FUNCTION_BLOCK FB_LowerFeedInConveyor EXTENDS FB_ActionBasic
VAR_INPUT
    xExecute    : BOOL;
    xAbort      : BOOL;
	xReset		: BOOL;
    Cylinder 	: REFERENCE TO UNI_CylinderList;
    TimeOut  	: LREAL := 30; // Unit : s
	Input		: ST_InputTable;
	OutPut		: ST_OutputTable;
	Motor		: REFERENCE TO UNI_MotorList;
END_VAR	
VAR_OUTPUT
    xAborted : BOOL;
    iErrorID : INT;
    ErrorMsg : T_MaxString;
END_VAR
VAR
    StateBehaviour   : CBML.ETrigATo;
    CurrentPosition : ST_PositionTable;
	uiCyclicStep    : UINT := 0;
	Reset_Rtrig 	:R_TRIG;
	
	TON_SensorDelay :TON;
	TON_ArrivedTimeOut :TON;
	TON_TimeOut :TON;
	fbExecuteEdgeDetect :FB_EdgeDetect;
END_VAR

THIS^.IBehaviourModel := StateBehaviour;
StateBehaviour(xExecute := xExecute,
              xAbort := xAbort OR fbExecuteEdgeDetect.xFallingEdge,
              udiTimeOut := LREAL_TO_UDINT( TimeOut*1000000),
              xDone => xDone,
              xBusy => xBusy,
              xError => xError,
              xAborted => xAborted);
//Error Mes
iErrorID := StateBehaviour._model.iErrorID;
ErrorMsg := M_GetErrorMsg(xErrorID := iErrorID);  

//Make sure that C# turns off execute to shut down the service
fbExecuteEdgeDetect(xInput :=xExecute);

//Reset 
Reset_Rtrig(CLK:= xReset);
IF Reset_Rtrig.Q THEN
	StateBehaviour.ResetModel(xCommit:=xReset);
END_IF

//Action
A00_BaseUnits();

ACTION A00_BaseUnits:
TON_SensorDelay(PT:= T#500MS);
TON_ArrivedTimeOut(PT:=T#30S);
TON_TimeOut(PT:=T#10S);
END_ACTION

METHOD CleanupAction
VAR_INPUT
    xAbortProposed : BOOL;
    iErrorIDProposed: INT;
END_VAR
VAR_OUTPUT
    xComplete : BOOL := TRUE;
    xAbort: BOOL := xAbortProposed;
 	iErrorID : INT := iErrorIDProposed;
END_VAR
END_METHOD

METHOD CyclicAction
VAR_INPUT
    itfTimingController : CBML.ITimingController;
END_VAR
VAR_OUTPUT
    xComplete : BOOL := TRUE;
    iErrorID : INT := 0;
END_VAR
xComplete :=FALSE;

CASE uiCyclicStep OF 
	
	100:	//檔盒上升， 呼叫輸送帶
		TON_TimeOut.IN:= TRUE;
		Cylinder.List.fbLowCV_Block2.M_Extend();
		IF Cylinder.List.fbLowCV_Block2.InFrontPosition THEN
			TON_TimeOut.IN:=FALSE;
			Motor.List.LowCV.M_MoveForward();
			uiCyclicStep:=150;
		END_IF
		IF TON_TimeOut.Q THEN 
			iErrorID :=10;
		END_IF
	150:	//check motor forward
		TON_TimeOut.IN :=TRUE;
		IF Motor.List.LowCV.InForWard THEN 
			TON_TimeOut.IN:=FALSE;
			uiCyclicStep:=200;
		END_IF
		IF TON_TimeOut.Q THEN
			iErrorID :=11;
		END_IF
	
	200:	//盒子到位, 延遲訊號,
		TON_ArrivedTimeOut.IN:= TRUE;
		TON_SensorDelay.IN := Input.bLowCV_Block2Detect_Sensor;
		IF TON_SensorDelay.Q THEN
			TON_SensorDelay.IN:=FALSE;
			TON_ArrivedTimeOut.IN:=FALSE;
			Cylinder.List.fbLowCV_Press4.M_Extend();
			uiCyclicStep:=300;
		END_IF
		IF TON_ArrivedTimeOut.Q THEN
			iErrorID :=9;
		END_IF
		
	300:	//檔盒下 等待第一盒到達最前sensor
		TON_TimeOut.IN:=TRUE;
		IF Cylinder.List.fbLowCV_Press4.InFrontPosition THEN
			Cylinder.List.fbLowCV_Block2.M_Retract();
		END_IF
		IF Cylinder.List.fbLowCV_Block2.InRearPosition THEN
			TON_TimeOut.IN:=FALSE;
			uiCyclicStep:=400;	
		END_IF
		IF TON_TimeOut.Q THEN
			iErrorID :=11;
		END_IF
		
	400:	//確認到最前sensor 
		TON_SensorDelay.IN:=Input.bLowCV_BoxArrived_Sensor;
		IF TON_SensorDelay.Q THEN
			TON_SensorDelay.IN:=FALSE;
			Cylinder.List.fbLowCV_Block2.M_Extend();
			uiCyclicStep:=500;
		END_IF
	
	500:	//釋放第二盒 
		IF 	Cylinder.List.fbLowCV_Block2.InFrontPosition THEN
			Cylinder.List.fbLowCV_Press4.M_Retract();
			uiCyclicStep:=600;
		END_IF
	600:	// 第二盒到檔盒位 第三盒壓盒檔上
		TON_SensorDelay.IN:= Input.bLowCV_Block2Detect_Sensor;
		IF TON_SensorDelay.Q THEN
			TON_SensorDelay.IN :=FALSE;
			Cylinder.List.fbLowCV_Press4.M_Extend();
			uiCyclicStep:= 700;
		END_IF
	
	700:	//釋放第二盒
		IF Cylinder.List.fbLowCV_Press4.InFrontPosition THEN
			Cylinder.List.fbLowCV_Block2.M_Retract();
			Cylinder.List.fbLowCV_Block1.M_Extend();
		END_IF
		IF Cylinder.List.fbLowCV_Block2.InRearPosition AND 
			Cylinder.List.fbLowCV_Block1.InFrontPosition THEN
			uiCyclicStep:= 800;
		END_IF
		
	800:	// 等待第二盒到夾盒位
		TON_SensorDelay.IN:=Input.bLowCV_Block1Detect_Sensor;
		IF TON_SensorDelay.Q THEN
			TON_SensorDelay.IN:=FALSE;
			Motor.List.LowCV.M_MotorStop();
			uiCyclicStep:=900;
		END_IF
	900:	//馬達停止 第一第二盒壓盒上
		IF Motor.List.LowCV.InStopped THEN
			Cylinder.List.fbLowCV_Press1.M_Extend();
			Cylinder.List.fbLowCV_Press2.M_Extend();
			Cylinder.List.fbLowCV_Block1.M_Retract();
			uiCyclicStep :=1000;
		END_IF
	1000:	//壓盒下
		IF Cylinder.List.fbLowCV_Press1.InFrontPosition AND 
			Cylinder.List.fbLowCV_Press2.InFrontPosition AND 
			Cylinder.List.fbLowCV_Block1.InRearPosition THEN
			Cylinder.List.fbLowCV_Press1.M_Retract();
			Cylinder.List.fbLowCV_Press2.M_Retract();
		END_IF
	1100:	//確認壓盒位置 回done
		IF Cylinder.List.fbLowCV_Press1.InRearPosition AND 
			Cylinder.List.fbLowCV_Press2.InRearPosition THEN 
			xComplete :=TRUE;
		END_IF
END_CASE
END_METHOD

METHOD ExitAction
VAR_INPUT
    xAfterCleanup : BOOL;
    xInCopyCode : BOOL;
END_VAR
TON_SensorDelay.IN:=FALSE;
END_METHOD

METHOD M_GetErrorMsg : T_MaxString
VAR_INPUT
	xErrorID: INT;
END_VAR

VAR
	
END_VAR
CASE xErrorID OF
	0:
		M_GetErrorMsg := 'No Error';
	1:
		M_GetErrorMsg := 'FB_LowerFeedInConveyor ErrorID 1: Action time out';
	2:
		M_GetErrorMsg := 'FB_LowerFeedInConveyor ErrorID 2: Position Data invalid';
	3:
		M_GetErrorMsg := 'FB_LowerFeedInConveyor ErrorID 3: LowCV_Block1 has Error in StartAction ';
	4:
		M_GetErrorMsg := 'FB_LowerFeedInConveyor ErrorID 4: LowCV_Block2 has Error in StartAction';
	5:
		M_GetErrorMsg := 'FB_LowerFeedInConveyor ErrorID 5: LowCV_Press1 has Error in StartAction';
	6:
		M_GetErrorMsg := 'FB_LowerFeedInConveyor ErrorID 6: LowCV_Press2 has Error in StartAction';
	7:
		M_GetErrorMsg := 'FB_LowerFeedInConveyor ErrorID 7: fbLowCV_Press3 has Error in StartAction';
	8:
		M_GetErrorMsg := 'FB_LowerFeedInConveyor ErrorID 8: fbLowCV_Press4 has Error in StartAction';
	9:
		M_GetErrorMsg := 'FB_LowerFeedInConveyor ErrorID 9: Box Arrived Time out not on LowCVBlock2' ;
	10:
		M_GetErrorMsg := 'FB_LowerFeedInConveyor ErrorID 10: Cylinder Error in CyclicAction';
	11:
		M_GetErrorMsg := 'FB_LowerFeedInConveyor ErrorID 11: Motor Error in CyclicAction';
									
		
		
		
		
END_CASE
END_METHOD

METHOD ResetAction
VAR_OUTPUT
    xComplete : BOOL := TRUE;
END_VAR
END_METHOD

METHOD StartAction
VAR_OUTPUT
    xComplete : BOOL := TRUE;
	iErrorID : INT := 0;
END_VAR
xComplete :=FALSE;

TON_SensorDelay.IN:=FALSE;

IF Cylinder.List.fbLowCV_Block1.xError THEN
	iErrorID := 3;
END_IF
IF Cylinder.List.fbLowCV_Block2.xError THEN
	iErrorID := 4;
END_IF
IF Cylinder.List.fbLowCV_Press1.xError THEN
	iErrorID := 5;
END_IF
IF Cylinder.List.fbLowCV_Press2.xError THEN
	iErrorID := 6;
END_IF
IF Cylinder.List.fbLowCV_Press3.xError THEN
	iErrorID := 7;
END_IF
IF Cylinder.List.fbLowCV_Press4.xError THEN
	iErrorID := 8;
END_IF

IF Cylinder.List.fbLowCV_Block1.InRearPosition AND
	Cylinder.List.fbLowCV_Block2.InRearPosition AND 
	Cylinder.List.fbLowCV_Press1.InRearPosition AND 
	Cylinder.List.fbLowCV_Press2.InRearPosition AND 
	Cylinder.List.fbLowCV_Press3.InRearPosition AND 
	Cylinder.List.fbLowCV_Press4.InRearPosition AND 
	Input.bLowCV_2ndBoxGap_Sensor THEN	//reverse logic sensor ,do make sure no box here 
	xComplete :=TRUE;
END_IF
END_METHOD

END_FUNCTION_BLOCK

(* stored: Version 1.1.0.1, ProductVersion 3.1.4024.13
   POU FB_LowerFeedInConveyor: Id {5557469c-d97a-40d7-bb66-ecb3bf04945c}, SpecialFunc None
   Folder Action: Id {f5856412-dfb9-4fb4-b243-7971692074bb}
   Action A00_BaseUnits: Id {434e8967-4fd8-4058-924a-a11daddc7b45}
   Method CleanupAction: Id {3ec3a4b0-0d7f-4322-b10b-b786adcf1a42}
   Method CyclicAction: Id {f1645a9f-a0da-4f2c-bba8-1031ddfe8693}
   Method ExitAction: Id {d057ae92-e162-415f-951a-6900793738e9}
   Method M_GetErrorMsg: Id {e76159c4-33a5-4234-a15a-b5dc4c12c867}
   Method ResetAction: Id {99fe9777-c7c6-45ea-a666-49c22fa3e079}
   Method StartAction: Id {3869020d-6432-4cf6-ac84-2285162f0a11} *)
